FUNCTION_BLOCK TF_Model (* Basic Function Block Type *)
  (* Standard: 61499-2 *)
  (* Version 0.3, 2009-09-15, JHC, Holobloc Inc, Changed transition priorities. *)
  (* Version 0.2, 2003-12-04, JHC, Rockwell Automation, Renamed for better indexing. *)
  (* Version 0.1, 2002-11-05, JHC, Rockwell Automation, Corrected missing ST element in Algorithm REQ. *)
  (* Version 0.0, 2000-05-30, JHC, Rockwell Automation *)
  PACKAGE fb.rt.mfb;
  IMPORT fb.datatype.*;
  IMPORT fb.rt.*;
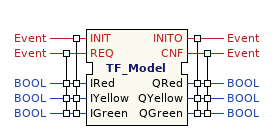
  EVENT_INPUT
    INIT WITH IRed, IYellow, IGreen; (* Initialization Request *)
    REQ WITH IRed, IYellow, IGreen; (* Normal Execution Request *)
  END_EVENT
  EVENT_OUTPUT
    INITO WITH QRed, QYellow, QGreen; (* Initialization Confirm *)
    CNF WITH QRed, QYellow, QGreen; (* Execution Confirmation *)
  END_EVENT
  VAR_INPUT
    IRed : BOOL; (* Input event qualifier *)
    IYellow : BOOL;
    IGreen : BOOL;
  END_VAR
  VAR_OUTPUT
    QRed : BOOL;
    QYellow : BOOL;
    QGreen : BOOL;
  END_VAR
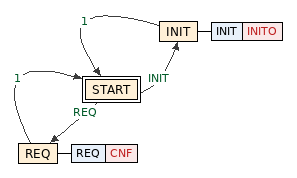
  EC_STATES
    START; (* Initial State *)
    INIT : INIT -> INITO; (* Initialization *)
    REQ : REQ -> CNF; (* Normal execution *)
  END_STATES
  EC_TRANSITIONS
    INIT TO START := 1;
    START TO REQ := REQ;
    START TO INIT := INIT;
    REQ TO START := 1;
  END_TRANSITIONS
  ALGORITHM INIT IN ST: (* Initialization algorithm *)

  END_ALGORITHM
  ALGORITHM REQ IN ST: (* Normally executed algorithm *)
QRed := IRed;
QYellow := IYellow;
QGreen := IGreen;
  END_ALGORITHM
END_FUNCTION_BLOCK
